{attribute 'GeneratedUsingTerminal: EK1100-0000-0018'}
{attribute addProperty BoxType "EK1100-0000-0018"}
{attribute addProperty Id "RH_A2_EK1122RH_A2_EK1122_10728E0974RH_A3_EL6631EL6631_A0EC075C2RH_A4_EL1809EL1809_32157CFD20RH_A5_EL1809EL1809_32157CFD20RH_A6_EL1809EL1809_32157CFD20RH_A7_EL2809EL2809_2B6483BD19RH_A8_EL1809EL1809_32157CFD20RH_A9_EL2809EL2809_2B6483BD19RH_A10_EL2809EL2809_2B6483BD19RH_A11_EL2809EL2809_2B6483BD19RH_EndTerminal_EL9011EL9011_D65D3D320"}
{attribute addProperty CRC "2777943550"}
{attribute addProperty Size "232"}
{attribute addProperty Name "RH (EK1100)"}
TYPE RH_EK1100_A5940DFE EXTENDS EK1100_1FC0878B :
STRUCT
	{attribute addProperty Name "RH_A2 (EK1122)"}
	{attribute addProperty PreviousPort "RH (EK1100) : B"}
	RH_A2_EK1122 : RH_A2_EK1122_10728E09;
	{attribute addProperty Name "RH_A3 (EL6631)"}
	{attribute addProperty PreviousPort "RH_A2 (EK1122) : C"}
	RH_A3_EL6631 : EL6631_A0EC075C;
	{attribute addProperty Name "RH_A4 (EL1809)"}
	{attribute addProperty PreviousPort "RH_A3 (EL6631) : B"}
	RH_A4_EL1809 : EL1809_32157CFD;
	{attribute addProperty Name "RH_A5 (EL1809)"}
	{attribute addProperty PreviousPort "RH_A4 (EL1809) : B"}
	RH_A5_EL1809 : EL1809_32157CFD;
	{attribute addProperty Name "RH_A6 (EL1809)"}
	{attribute addProperty PreviousPort "RH_A5 (EL1809) : B"}
	RH_A6_EL1809 : EL1809_32157CFD;
	{attribute addProperty Name "RH_A7 (EL2809)"}
	{attribute addProperty PreviousPort "RH_A6 (EL1809) : B"}
	RH_A7_EL2809 : EL2809_2B6483BD;
	{attribute addProperty Name "RH_A8 (EL1809)"}
	{attribute addProperty PreviousPort "RH_A7 (EL2809) : B"}
	RH_A8_EL1809 : EL1809_32157CFD;
	{attribute addProperty Name "RH_A9 (EL2809)"}
	{attribute addProperty PreviousPort "RH_A8 (EL1809) : B"}
	RH_A9_EL2809 : EL2809_2B6483BD;
	{attribute addProperty Name "RH_A10 (EL2809)"}
	{attribute addProperty PreviousPort "RH_A9 (EL2809) : B"}
	RH_A10_EL2809 : EL2809_2B6483BD;
	{attribute addProperty Name "RH_A11 (EL2809)"}
	{attribute addProperty PreviousPort "RH_A10 (EL2809) : B"}
	RH_A11_EL2809 : EL2809_2B6483BD;
	{attribute addProperty Name "RH_EndTerminal (EL9011)"}
	{attribute addProperty PreviousPort "RH_A11 (EL2809) : B"}
	RH_EndTerminal_EL9011 : EL9011_D65D3D32;
END_STRUCT
END_TYPE

(* stored: Version 1.2.0.0, ProductVersion 3.1.4024.11
   DUT RH_EK1100_A5940DFE: Id {d591c9a6-6b1a-0794-18dc-d8e405ad3b6a} *)
